TYPE EL5042_Status : ST_EL5042_Status; END_TYPE

(* stored: Version 1.1.0.1, ProductVersion 3.1.4022.18
   DUT EL5042_Status: Id {8d65cae0-9efe-4c5b-a7a7-f17022f98dd4} *)
